FUNCTION_BLOCK FB_ADSLOG_reporter IMPLEMENTS InterfaceJobEventReporter
VAR_INPUT
END_VAR
VAR_OUTPUT
	text : T_MAXSTRING;
END_VAR
VAR
END_VAR

{warning 'add method implementation '}
METHOD report : BOOL
VAR_INPUT
	old_state	: E_FutureExecutionState;
	new_state	: E_FutureExecutionState;
	record_time	: Tc2_Utilities.T_FILETIME64;
	executor	: REFERENCE TO FB_Executor;
END_VAR
VAR_INST
	fb_timezone_info : FB_GetTimeZoneInformation := (bExecute := TRUE);
END_VAR
VAR
	last_state : STRING;
	current_state : STRING;
END_VAR
last_state := TO_STRING(old_state);
current_state := TO_STRING(new_state);
fb_timezone_info();
text := FILETIME64_TO_ISO8601(fileTime := record_time, nBias := DINT_TO_INT(fb_timezone_info.tzInfo.bias), bUTC := TRUE,nPrecision := 6);
text := CONCAT(text, ':');
text := CONCAT(text, last_state);
text := CONCAT(text, '->');
text := CONCAT(text, TO_STRING(current_state));
text := CONCAT(text, ':');
text := CONCAT(text, executor.future.future_name);
text := CONCAT(text, ':');
text := CONCAT(text, '%s');

ADSLOGSTR(msgCtrlMask := ADSLOG_MSGTYPE_LOG, msgFmtStr := text, strArg := executor.id);

report := TRUE;
END_METHOD

END_FUNCTION_BLOCK

(* stored: Version 1.1.0.1, ProductVersion 3.1.4024.12
   POU FB_ADSLOG_reporter: Id {ba91026f-1b14-496b-9bee-5db4c9acb690}, SpecialFunc None
   Method report: Id {e5fac08e-bd79-4abd-97a0-a76262921e4d} *)
